// TIA Portal V19 export
TYPE "PPrg_Data"
// stored: Access Published
   STRUCT
      Header { S7_SetPoint := 'True'} : "Prg_Header";
   END_STRUCT;
END_TYPE
